Staubli VAL3: Simulation.dtx

mdesc mNomSpeed
sio sSocket = {link=Socket\Feedback}
tool tToolSuccion = {z=110, fatherId=flange[0], ioLink=valve2}
num nConnection
num nRecvData
jointRx JApproach1 = {j2=9, j3=75, j5=93, j6=142}
jointRx JHome = {j3=0.6}
screen sMonitor
num l_nRetVal
pointRx pApprBins = {x=451, y=82, z=170, rx=-178, rz=-39, fatherId=world[0]}
pointRx pBinYellow = {x=539, y=-98, z=11, rx=-178, rz=-39, fatherId=world[0]}
pointRx pBinBlue = {x=346, y=-101, z=10, rx=-178, rz=-39, fatherId=world[0]}
pointRx pBinGreen = {x=542, y=233, z=10, rx=-178, rz=-39, fatherId=world[0]}
pointRx pBinBrown = {x=346, y=180, z=11, rx=-178, rz=-39, fatherId=world[0]}
jointRx jGetCinta = {j1=-88, j2=71, j3=56, j5=53, j6=50}
bool bStop
num nkey
jointRx jAproachCinta = {j1=-82, j2=60, j3=56.5, j5=65, j6=50}
pointRx pTable = {x=256.13, y=-12.37, z=50, rx=-178, rz=-39, fatherId=world[0]}
tool tToolGripper = {z=115, fatherId=flange[0], ioLink=valve1}
sio sPlc = {link=Socket\PLClient}
num nRecvPLC
jointRx jGetPaperCinta = {j1=-94, j2=83, j3=43, j5=56}
jointRx jGetPlaGlaCinta = {j1=-93, j2=73, j3=54, j5=55}
jointRx jBinGreen = {j1=16, j2=62, j3=30, j5=88, j6=157}
jointRx jBinYellow = {j1=-13, j2=56, j3=41, j5=84, j6=127}
bool bChangeTool
string sTecla
jointRx jChangeTool = {j1=80, j2=45, j3=64, j5=34, j6=52}
